Fanuc KAREL source: KT00139.KL

PROGRAM KT00139
%NOLOCKGROUP
VAR
  R1: REAL
  R2: REAL
  OUT: INTEGER
BEGIN
  R1 = 2.0
  R2 = 3.0
  R1 = 2.0
  R2 = 3.0
  OUT = R1 DIV R2
END KT00139
